PROGRAM pouMcAlarms
VAR
	idbMsgAlarm: FB_CheckMessageBounds;
END_VAR

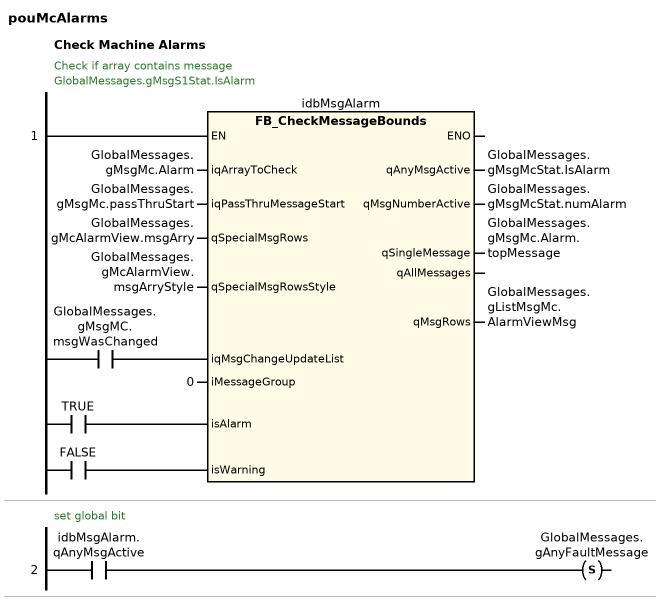
// NETWORK 1: Check Machine Alarms
// Check if array contains message
//
// GlobalMessages.gMsgS1Stat.IsAlarm
idbMsgAlarm(
    iqArrayToCheck := GlobalMessages.gMsgMc.Alarm,
    iqPassThruMessageStart := GlobalMessages.gMsgMc.passThruStart,
    qSpecialMsgRows := GlobalMessages.gMcAlarmView.msgArry,
    qSpecialMsgRowsStyle := GlobalMessages.gMcAlarmView.msgArryStyle,
    iqMsgChangeUpdateList := GlobalMessages.gMsgMC.msgWasChanged,
    iMessageGroup := 0,
    isAlarm := TRUE,
    isWarning := FALSE,
    qAnyMsgActive => GlobalMessages.gMsgMcStat.IsAlarm,
    qMsgNumberActive => GlobalMessages.gMsgMcStat.numAlarm,
    qSingleMessage => GlobalMessages.gMsgMc.Alarm.topMessage,
    qMsgRows => GlobalMessages.gListMsgMc.AlarmViewMsg); // FB_CheckMessageBounds

// NETWORK 2
// set global bit
GlobalMessages.gAnyFaultMessage S= idbMsgAlarm.qAnyMsgActive;

END_PROGRAM

(* stored: Version 1.1.0.1, ProductVersion 3.1.4024.11
   POU pouMcAlarms: Id {3f0fd1a1-2fbb-4f59-9ec9-208cf01105f8}, SpecialFunc None *)
